// TIA Portal V19 export
ORGANIZATION_BLOCK "Sim"   // OB124, FBD, ProgramCycle
TITLE = "Main Program Sweep (Cycle)"
{ S7_Optimized_Access := 'TRUE' }
// stored: SetENOAutomatically false
   VAR_INPUT
      Initial_Call : Bool;   // Initial call of this OB
      Remanence : Bool;   // =True, if remanent data are available
   END_VAR
BEGIN

REGION Network 1
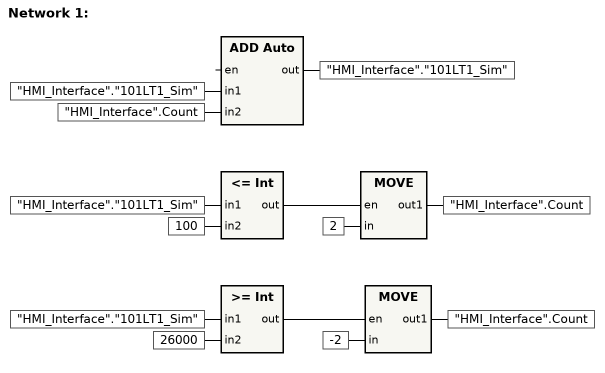
   "HMI_Interface"."101LT1_Sim" := "HMI_Interface"."101LT1_Sim" + "HMI_Interface".Count;
   IF "HMI_Interface"."101LT1_Sim" <= 100 THEN "HMI_Interface".Count := 2; END_IF;
   IF "HMI_Interface"."101LT1_Sim" >= 26000 THEN "HMI_Interface".Count := -2; END_IF;
END_REGION
END_ORGANIZATION_BLOCK
